Staubli VAL3: IF.dtx

string sChoice[4]
  [0] = "IN"
  [1] = "OUT"
  [3] = "NUM"
public string sItems
string sMessage
